FUNCTION F_MathTest : LREAL
VAR_INPUT
	fA : LREAL;
	fB : LREAL;
END_VAR
VAR
END_VAR

F_MathTest := fA + fB;

END_FUNCTION

(* stored: Version 1.1.0.1, ProductVersion 3.1.4024.10
   POU F_MathTest: Id {b2e980b4-d02a-4279-a1c3-2d21b12e9815}, SpecialFunc None *)
